(* PLC project Tc2_Utilities.Profiler Demo, tc3-libraries-kb TwinCAT 3.1 *)
(* stored: creationDateTime 2026-05-11T00:00:00, modificationDateTime 2026-05-11T00:00:00 *)

PROGRAM P_Demo_Profiler
  VAR
    fbProfiler : Profiler;  (* Profiler 实例 *)
    START : BOOL;
    RESET : BOOL;
    BUSY : BOOL;
    DATA : PROFILERSTRUCT;
  END_VAR

// =============================================================================
// 场景：优化对比。
// 价值：定位热点。
// 验证：Start → 业务代码 → Stop → 读 nElapsed 微秒值。
// 验证步骤：
//   1. 右键 PLC 项目 → Import PLCopenXML → 选本文件
//   2. 引用 Tc2_Utilities（References → Add library）
//   3. 编译 → 登录 → 运行；按上方『验证』行的指示在线写值观察
// =============================================================================

// 单次完整调用形式（所有 VAR_INPUT 显式赋值）
fbProfiler(
    START := START,
    RESET := RESET,
    BUSY => BUSY,
    DATA => DATA
);
END_PROGRAM
